TYPE SharedContextComPublish :
STRUCT
  Region1 : ZApplication.RegionComPublish;
  Region2 : ZApplication.RegionComPublish;
  Region3 : ZApplication.RegionComPublish;
  Region4 : ZApplication.RegionComPublish;
  Region5 : ZApplication.RegionComPublish;
  Region6 : ZApplication.RegionComPublish;
  Region7 : ZApplication.RegionComPublish;
END_STRUCT
END_TYPE

(* stored: Version 1.1.0.1
   DUT SharedContextComPublish: Id {60aa59be-fb66-4e61-9e8b-b545b7efc5ab} *)
